Yaskawa INFORM job: M004SDP.JBI

/JOB
//NAME M004SDP
//POS
///NPOS 0,0,0,0,0,0
//INST
///DATE 2019/08/05 22:05
///ATTR SC,RW,MC
///GROUP1 RB1
///LVARS 0,0,3,0,0,0,0,0
NOP
GETARG LD000 IARG#(1)
GETARG LD001 IARG#(2)
SET D070 LD000
SET D071 LD001
SET B069 0
SKILLSND "Comm004SendPos"
WAIT B069=1
END
